PROGRAM MAIN
VAR
	
END_VAR

// copio i 16 bit di ingresso sulle 16 linee di uscita
GVL_IO.DQ := GVL_IO.DI;

END_PROGRAM

(* stored: Version 1.1.0.1
   POU MAIN: Id {d6a97a93-bbbb-4808-8334-637627ec2e0f}, SpecialFunc None *)
